PROGRAM Hoofdschakelaar_
VAR
	 Step: UINT:=0; 
END_VAR


    // Hoofdschakelaar is true, turn on the lamp
   
        IF GVL.Hoofdschakelaar THEN
            GVL.Lamp_Hoofdschakelaar := TRUE;
		 ELSE
            GVL.Lamp_Hoofdschakelaar := FALSE;
        END_IF;

END_PROGRAM

(* stored: Version 1.1.0.1, ProductVersion 3.1.4024.12
   POU Hoofdschakelaar_: Id {6f2732b7-697e-4cb4-b219-cb190d32e081}, SpecialFunc None *)
